(* IEC 61131-3 sources: F100R_S278_Temperville/MyController.device.xml.v3^/Plc Logic.plclogic.xml.v3^/Application.application.xml.v3^/00_FB, 42 files *)

(* ---- Valor_Float.fn.st ---- *)
FUNCTION Valor_Float : REAL
VAR_INPUT
	Input_01: WORD;
	Input_02: WORD;
END_VAR
VAR
	Convert_01: WORD_AS_DWORD;
	DW_AxOutpt: DWORD;
	Bit_DWord_Mantissa: BIT_AS_DWORD;
	Aux_Mantissa: DWORD;
	Mantissa1: REAL;
	Bit_DW_Expoente: BIT_AS_DWORD;
	Aux_Exp: DWORD;
	Aux_Exp2: REAL;
	Expoente: REAL;
	Sinal: REAL;
	Sinal2: REAL;
	base1: REAL;
END_VAR

Convert_01(i_wLow:= Input_01, i_wHigh:= Input_02, q_dwOput=>DW_AxOutpt );

(*=========== F=-1^s * 2^(e-127) * (1 + M/2^23)============= *)

//Composição da Mantissa
Bit_DWord_Mantissa(
	B00:= DW_AxOutpt.0,
	B01:= DW_AxOutpt.1,
	B02:= DW_AxOutpt.2,
	B03:= DW_AxOutpt.3,
	B04:= DW_AxOutpt.4,
	B05:= DW_AxOutpt.5,
	B06:= DW_AxOutpt.6,
	B07:= DW_AxOutpt.7,
	B08:= DW_AxOutpt.8,
	B09:= DW_AxOutpt.9,
	B10:= DW_AxOutpt.10,
	B11:= DW_AxOutpt.11,
	B12:= DW_AxOutpt.12,
	B13:= DW_AxOutpt.13,
	B14:= DW_AxOutpt.14,
	B15:= DW_AxOutpt.15,
	B16:= DW_AxOutpt.16,
	B17:= DW_AxOutpt.17,
	B18:= DW_AxOutpt.18,
	B19:= DW_AxOutpt.19,
	B20:= DW_AxOutpt.20,
	B21:= DW_AxOutpt.21,
	B22:= DW_AxOutpt.22,
	X=> Aux_Mantissa);

	Mantissa1:= DWORD_TO_REAL (Aux_Mantissa);

	//Composição Expoente

	Bit_DW_Expoente(
	B00:= DW_AxOutpt.23,
	B01:= DW_AxOutpt.24,
	B02:= DW_AxOutpt.25,
	B03:= DW_AxOutpt.26,
	B04:= DW_AxOutpt.27,
	B05:= DW_AxOutpt.28,
	B06:= DW_AxOutpt.29,
	B07:= DW_AxOutpt.30,
	X=> Aux_Exp);

	Aux_Exp2:= DWORD_TO_REAL (Aux_Exp - 127);

	Expoente:= EXPT (2,Aux_Exp2);

	//Sinal
	base1:=BOOL_TO_REAL (DW_AxOutpt.31);
	Sinal2:= EXPT (-1,base1);

	// Equação para o resultado em FLOAT

	Valor_Float:= Sinal2 * Expoente * (1 + Mantissa1/ 8388608);

(* ---- AlarmeEncoder.fb.st ---- *)
FUNCTION_BLOCK AlarmeEncoder
VAR_INPUT
	xHabilitaAlarme: BOOL;
	xResetAlarme: BOOL;
	ixCanalA: BOOL;
	ixCanalB: BOOL;
	tTempoPulso: TIME;
END_VAR
VAR_OUTPUT
	xAlarmeCanalA: BOOL;
	xAlarmeCanalB: BOOL;
	xAlarmeGeral: BOOL;
	xAlarmeSonoro: BOOL;
END_VAR
VAR
	TonAtrasoAlarme: TON;
	TonAtrasoAlarmeIn: BOOL;
	TonAtrasoAlarmePt: TIME;
	TonAtrasoAlarmeQ: BOOL;
	TonPulsoCanalAUp: TON;
	TonPulsoCanalAUpIn: BOOL;
	TonPulsoCanalAUpPt: TIME;
	TonPulsoCanalAUpQ: BOOL;
	TonPulsoCanalADown: TON;
	TonPulsoCanalADownIn: BOOL;
	TonPulsoCanalADownPt: TIME;
	TonPulsoCanalADownQ: BOOL;
	TonPulsoCanalBUp: TON;
	TonPulsoCanalBUpIn: BOOL;
	TonPulsoCanalBUpPt: TIME;
	TonPulsoCanalBUpQ: BOOL;
	TonPulsoCanalBDown: TON;
	TonPulsoCanalBDownIn: BOOL;
	TonPulsoCanalBDownPt: TIME;
	TonPulsoCanalBDownQ: BOOL;
	TonSinAlarme: TON;
	TonSinAlarmeIn: BOOL;
	TonSinAlarmePt: TIME;
	TonSinAlarmeQ: BOOL;
	TpSireneAlarme: TP;
	TpSireneAlarmeIn: BOOL;
	TpSireneAlarmePt: TIME;
	TpSireneAlarmeQ: BOOL;
	xHabilitadorMonitoraAlarme: BOOL;
END_VAR

(*Bloco de Monitoramento de Encoder pelas Entradas Digitais*)

(*---- Habilita Monitoramento de Alarme de Defeito ----*)
if xHabilitaAlarme then
	TonAtrasoAlarmeIn:=true;
else
	TonAtrasoAlarmeIn:=false;
end_if;

(*--- Tempo de Atraso para Inicio do Monitoramento ---*)
TonAtrasoAlarme (IN := TonAtrasoAlarmeIn,
		 PT := T#1500ms,
                 Q => TonAtrasoAlarmeQ);

xHabilitadorMonitoraAlarme:=TonAtrasoAlarmeQ;

(*--- Monitoramento do Canal A ---*)
(*--- Canal A Defeito Alto ---*)
TonPulsoCanalAUpIn:=xHabilitadorMonitoraAlarme and not ixCanalA;

TonPulsoCanalAUp (IN := TonPulsoCanalAUpIn,
                PT :=  tTempoPulso,
                Q => TonPulsoCanalAUpQ);

(*--- Canal A Defeito Baixo ---*)
TonPulsoCanalADownIn:=xHabilitadorMonitoraAlarme and ixCanalA;

TonPulsoCanalADown (IN := TonPulsoCanalADownIn,
                PT := tTempoPulso,
                Q => TonPulsoCanalADownQ);

(*--- Alarme Defeito Canal A ---*)

if TonPulsoCanalAUpQ or TonPulsoCanalADownQ then
	xAlarmeCanalA:=true;
end_if;

(*--------------------------------*)
(*--- Monitoramento do Canal B ---*)
(*--- Canal B Defeito Alto ---*)
TonPulsoCanalBUpIn:=xHabilitadorMonitoraAlarme and not ixCanalB;

TonPulsoCanalBUp (IN := TonPulsoCanalBUpIn,
                PT := tTempoPulso,
                Q => TonPulsoCanalBUpQ);

(*--- Canal A Defeito Baixo ---*)
TonPulsoCanalBDownIn:=xHabilitadorMonitoraAlarme and ixCanalB;

TonPulsoCanalBDown (IN := TonPulsoCanalBDownIn,
                PT := tTempoPulso,
                Q => TonPulsoCanalBDownQ);

(*--- Alarme Defeito Canal B ---*)

if TonPulsoCanalBUpQ or TonPulsoCanalBDownQ then
	xAlarmeCanalB:=true;
end_if;

(*--------------------------------*)
(*--- Indicação Alarme Geral ---*)
xAlarmeGeral:=xAlarmeCanalA or xAlarmeCanalB;

(*--- Alarme Sonoro ---*)
TpSireneAlarmeIn:=xAlarmeGeral;

TpSireneAlarme (IN := TpSireneAlarmeIn,
                PT := T#500ms,
                Q => TpSireneAlarmeQ);

if TpSireneAlarmeQ then
	xAlarmeSonoro:=true;
end_if;

(*--- Reseta Alarmes do Encoder ---*)
if xResetAlarme then
	xAlarmeCanalA:=false;
	xAlarmeCanalB:=false;
	xAlarmeSonoro:=false;
end_if;

(* ---- AlarmeMotor.fb.st ---- *)
FUNCTION_BLOCK AlarmeMotor
VAR_INPUT
	KaMotor: BOOL;
	KmMotor: BOOL;
	ResetAlarm: BOOL;
END_VAR
VAR_OUTPUT
	AlarmeMotor: BOOL;
	AlarmeSonoro: BOOL;
END_VAR
VAR
	TonAlarme: TON;
	TpSom: TP;
END_VAR

TonAlarme.IN:= KmMotor AND NOT KaMotor;

TonAlarme(PT:=T#100MS );

IF TonAlarme.Q THEN
	AlarmeMotor:= TRUE;
END_IF

TpSom(IN:= AlarmeMotor , PT:= T#500MS );

IF TpSom.Q THEN
	AlarmeSonoro:=TRUE;
END_IF

IF	ResetAlarm THEN
	AlarmeMotor:=FALSE;
	AlarmeSonoro:=FALSE;
END_IF

(* ---- AlarmeMotorParado.fb.st ---- *)
FUNCTION_BLOCK AlarmeMotorParado
VAR_INPUT
	KaMotor: BOOL;
	ResetAlarm: BOOL;
END_VAR
VAR_OUTPUT
	AlarmeMotor: BOOL;
	AlarmeSonoro: BOOL;
END_VAR
VAR
	TonAlarme: TON;
	TpSom: TP;
	TpReset: TP;
END_VAR

TonAlarme.IN:= KaMotor;

TonAlarme(PT:=T#3000MS );

IF TonAlarme.Q THEN
	AlarmeMotor:= TRUE;
END_IF

TpSom(IN:= AlarmeMotor , PT:= T#500MS );

IF TpSom.Q THEN
	AlarmeSonoro:=TRUE;
END_IF

TpReset(IN:= ResetAlarm , PT:= T#1000MS );

IF	TpReset.Q THEN
	AlarmeMotor:=FALSE;
	AlarmeSonoro:=FALSE;
END_IF

(* ---- AlarmeRelesSsr.fb.st ---- *)
FUNCTION_BLOCK AlarmeRelesSsr
VAR_INPUT
	RetornoReleSsr: BOOL;
	ResistRompida: BOOL;
	ReleSsr: BOOL;
	ResetAlarm: BOOL;
END_VAR
VAR_OUTPUT
	AlarmeSsrAberto: BOOL;
	AlarmeSsrFechado: BOOL;
	AlarmeSonoro: BOOL;
END_VAR
VAR
	TonAberto: TON;
	TonFechado: TON;
	TpSom: TP;
END_VAR

TonAberto.IN:= ReleSsr AND NOT RetornoReleSsr;
TonFechado.IN:= RetornoReleSsr AND NOT ResistRompida AND NOT ReleSsr;

TonAberto(PT:=T#400MS );
TonFechado(PT:=T#400MS );

IF TonAberto.Q THEN
	AlarmeSsrAberto:= TRUE;
END_IF

IF TonFechado.Q THEN
	AlarmeSsrFechado:=TRUE;
END_IF

TpSom(IN:= AlarmeSsrAberto OR AlarmeSsrFechado, PT:= T#200MS );

IF TpSom.Q THEN
	AlarmeSonoro:=TRUE;
END_IF

IF	ResetAlarm THEN
	AlarmeSsrAberto:=FALSE;
	AlarmeSsrFechado:=FALSE;
	AlarmeSonoro:=FALSE;
END_IF

(* ---- AlarmeResistencia.fb.st ---- *)
FUNCTION_BLOCK AlarmeResistencia
VAR_INPUT
	ResistRompida: BOOL;
	ResetAlarm: BOOL;
END_VAR
VAR_OUTPUT
	AlarmeResistRompida: BOOL;
	AlarmeSonoro: BOOL;
END_VAR
VAR
	TonRompida: TON;
	TpSom: TP;
END_VAR

TonRompida.IN:=ResistRompida;

TonRompida(PT:=T#250ms);

IF TonRompida.Q THEN
	AlarmeResistRompida:=TRUE;
END_IF

TpSom(IN:= AlarmeResistRompida, PT:= T#500MS);

IF TpSom.Q THEN
	AlarmeSonoro:=TRUE;
END_IF

IF	ResetAlarm THEN
	AlarmeResistRompida:=FALSE;
	AlarmeSonoro:=FALSE;
END_IF

(* ---- AlarmeTemperatura.fb.st ---- *)
FUNCTION_BLOCK AlarmeTemperatura
VAR_INPUT
	TermoparAtual: REAL;
	TemperaturaMax: REAL;
	ResetAlarm: BOOL;
END_VAR
VAR_OUTPUT
	TermoparAlmTemperatura: BOOL;
	AlarmeSonAlmTemperatura: BOOL;
END_VAR
VAR
	TonTh: TON;
	TpSom: TP;
	TemperaturaExcedeu: BOOL;
END_VAR

TemperaturaExcedeu:=(TermoparAtual >= TemperaturaMax);

TonTh.IN:=TemperaturaExcedeu;

TonTh(PT:=T#1S);

IF TonTh.Q THEN
	TermoparAlmTemperatura:=TRUE;
END_IF

TpSom(IN:=TermoparAlmTemperatura,PT:=T#1S);

IF TpSom.Q THEN
	AlarmeSonAlmTemperatura:=TRUE;
END_IF

IF	ResetAlarm THEN
	TermoparAlmTemperatura:=FALSE;
	AlarmeSonAlmTemperatura:=FALSE;
END_IF

(* ---- AlarmeTermopar.fb.st ---- *)
FUNCTION_BLOCK AlarmeTermopar
VAR_INPUT
	Termopar: BOOL;
	ResetAlarm: BOOL;
END_VAR
VAR_OUTPUT
	TermoparAberto: BOOL;
	AlarmeSonTermopar: BOOL;
END_VAR
VAR
	TonTh: TON;
	TpSom: TP;
END_VAR

TonTh.IN:=Termopar;

TonTh(PT:=T#1S);

IF TonTh.Q THEN
	TermoparAberto:=TRUE;
END_IF

TpSom(IN:=TermoparAberto,PT:=T#1S);

IF TpSom.Q THEN
	AlarmeSonTermopar:=TRUE;
END_IF

IF	ResetAlarm THEN
	TermoparAberto:=FALSE;
	AlarmeSonTermopar:=FALSE;
END_IF

(* ---- AlarmeTM3TI8T.fb.st ---- *)
FUNCTION_BLOCK AlarmeTM3TI8T
VAR_INPUT
	inAlarmeInput01: BYTE;
	inAlarmeInput02: BYTE;
	inAlarmeInput03: BYTE;
	inAlarmeInput04: BYTE;
	inAlarmeInput05: BYTE;
	inAlarmeInput06: BYTE;
	inAlarmeInput07: BYTE;
	inAlarmeInput08: BYTE;
END_VAR
VAR_OUTPUT
	OutAlarmeInput01: BOOL;
	OutAlarmeInput02: BOOL;
	OutAlarmeInput03: BOOL;
	OutAlarmeInput04: BOOL;
	OutAlarmeInput05: BOOL;
	OutAlarmeInput06: BOOL;
	OutAlarmeInput07: BOOL;
	OutAlarmeInput08: BOOL;
END_VAR
VAR
	TonTh01: TON;
	TonTh02: TON;
	TonTh03: TON;
	TonTh04: TON;
	TonTh05: TON;
	TonTh06: TON;
	TonTh07: TON;
	TonTh08: TON;
	xTermopar01Aberto: BOOL;
	xTermopar02Aberto: BOOL;
	xTermopar03Aberto: BOOL;
	xTermopar04Aberto: BOOL;
	xTermopar05Aberto: BOOL;
	xTermopar06Aberto: BOOL;
	xTermopar07Aberto: BOOL;
	xTermopar08Aberto: BOOL;
END_VAR

//TERMOPAR 01
IF inAlarmeInput01=5 OR inAlarmeInput01=6 OR inAlarmeInput01=4 THEN
	xTermopar01Aberto:=TRUE;
ELSE
	xTermopar01Aberto:=FALSE;
END_IF

//TERMOPAR 02
IF inAlarmeInput02=5 OR inAlarmeInput02=6 OR inAlarmeInput02=4 THEN
	xTermopar02Aberto:=TRUE;
ELSE
	xTermopar02Aberto:=FALSE;
END_IF

//TERMOPAR 03
IF inAlarmeInput03=5 OR inAlarmeInput03=6 OR inAlarmeInput03=4 THEN
	xTermopar03Aberto:=TRUE;
ELSE
	xTermopar03Aberto:=FALSE;
END_IF

//TERMOPAR 04
IF inAlarmeInput04=5 OR inAlarmeInput04=6 OR inAlarmeInput04=4 THEN
	xTermopar04Aberto:=TRUE;
ELSE
	xTermopar04Aberto:=FALSE;
END_IF

//TERMOPAR 05
IF inAlarmeInput05=5 OR inAlarmeInput05=6 OR inAlarmeInput05=4 THEN
	xTermopar05Aberto:=TRUE;
ELSE
	xTermopar05Aberto:=FALSE;
END_IF

//TERMOPAR 06
IF inAlarmeInput06=5 OR inAlarmeInput06=6 OR inAlarmeInput06=4 THEN
	xTermopar06Aberto:=TRUE;
ELSE
	xTermopar06Aberto:=FALSE;
END_IF

//TERMOPAR 07
IF inAlarmeInput07=5 OR inAlarmeInput07=6 OR inAlarmeInput07=4 THEN
	xTermopar07Aberto:=TRUE;
ELSE
	xTermopar07Aberto:=FALSE;
END_IF

//TERMOPAR 08
IF inAlarmeInput08=5 OR inAlarmeInput08=6 OR inAlarmeInput08=4 THEN
	xTermopar08Aberto:=TRUE;
ELSE
	xTermopar08Aberto:=FALSE;
END_IF

TonTh01(IN:=xTermopar01Aberto, PT:=T#0S , Q=>OutAlarmeInput01);
TonTh02(IN:=xTermopar02Aberto, PT:=T#0S , Q=>OutAlarmeInput02);
TonTh03(IN:=xTermopar03Aberto, PT:=T#0S , Q=>OutAlarmeInput03);
TonTh04(IN:=xTermopar04Aberto, PT:=T#0S , Q=>OutAlarmeInput04);
TonTh05(IN:=xTermopar05Aberto, PT:=T#0S , Q=>OutAlarmeInput05);
TonTh06(IN:=xTermopar06Aberto, PT:=T#0S , Q=>OutAlarmeInput06);
TonTh07(IN:=xTermopar07Aberto, PT:=T#0S , Q=>OutAlarmeInput07);
TonTh08(IN:=xTermopar08Aberto, PT:=T#0S , Q=>OutAlarmeInput08);

(* ---- AlarmeTM5SAI6TH.fb.st ---- *)
FUNCTION_BLOCK AlarmeTM5SAI6TH
VAR_INPUT
	bEntradaByte00: BYTE;
	bEntradaByte01: BYTE;
	ResetAlarm: BOOL;
END_VAR
VAR_OUTPUT
	Termopar01AbaixoMinimo: BOOL;
	Termopar01AcimaMaximo: BOOL;
	Termopar01Ok: BOOL;
	Termopar01Aberto: BOOL;
	Termopar02AbaixoMinimo: BOOL;
	Termopar02AcimaMaximo: BOOL;
	Termopar02Ok: BOOL;
	Termopar02Aberto: BOOL;
	Termopar03AbaixoMinimo: BOOL;
	Termopar03AcimaMaximo: BOOL;
	Termopar03Ok: BOOL;
	Termopar03Aberto: BOOL;
	Termopar04AbaixoMinimo: BOOL;
	Termopar04AcimaMaximo: BOOL;
	Termopar04Ok: BOOL;
	Termopar04Aberto: BOOL;
	Termopar05AbaixoMinimo: BOOL;
	Termopar05AcimaMaximo: BOOL;
	Termopar05Ok: BOOL;
	Termopar05Aberto: BOOL;
	Termopar06AbaixoMinimo: BOOL;
	Termopar06AcimaMaximo: BOOL;
	Termopar06Ok: BOOL;
	Termopar06Aberto: BOOL;
END_VAR
VAR
	StatusByte00: BYTE_AS_BIT;
	StatusByte01: BYTE_AS_BIT;
	xEntradaTermopar0101: BOOL;
	xEntradaTermopar0201: BOOL;
	xEntradaTermopar0102: BOOL;
	xEntradaTermopar0202: BOOL;
	xEntradaTermopar0103: BOOL;
	xEntradaTermopar0203: BOOL;
	xEntradaTermopar0104: BOOL;
	xEntradaTermopar0204: BOOL;
	xEntradaTermopar0105: BOOL;
	xEntradaTermopar0205: BOOL;
	xEntradaTermopar0106: BOOL;
	xEntradaTermopar0206: BOOL;
	TonTh01: TON;
	TonTh02: TON;
	TonTh03: TON;
	TonTh04: TON;
	TonTh05: TON;
	TonTh06: TON;
END_VAR

StatusByte00(
		B:= bEntradaByte00,
		B0=> xEntradaTermopar0101,
		B1=> xEntradaTermopar0201,
		B2=> xEntradaTermopar0102,
		B3=> xEntradaTermopar0202,
		B4=> xEntradaTermopar0103,
		B5=> xEntradaTermopar0203,
		B6=> xEntradaTermopar0104,
		B7=> xEntradaTermopar0204);

StatusByte01(
		B:= bEntradaByte01,
		B0=> xEntradaTermopar0105,
		B1=> xEntradaTermopar0205,
		B2=> xEntradaTermopar0106,
		B3=> xEntradaTermopar0206);

Termopar01Ok:= NOT xEntradaTermopar0101 AND NOT xEntradaTermopar0201;
Termopar01AbaixoMinimo:= NOT xEntradaTermopar0101 AND xEntradaTermopar0201;
Termopar01AcimaMaximo:= xEntradaTermopar0101 AND NOT xEntradaTermopar0201;
TonTh01.IN:= xEntradaTermopar0101 AND xEntradaTermopar0201;

Termopar02Ok:= NOT xEntradaTermopar0102 AND NOT xEntradaTermopar0202;
Termopar02AbaixoMinimo:= NOT xEntradaTermopar0102 AND xEntradaTermopar0202;
Termopar02AcimaMaximo:= xEntradaTermopar0102 AND NOT xEntradaTermopar0202;
TonTh02.IN:= xEntradaTermopar0102 AND xEntradaTermopar0202;

Termopar03Ok:= NOT xEntradaTermopar0103 AND NOT xEntradaTermopar0203;
Termopar03AbaixoMinimo:= NOT xEntradaTermopar0103 AND xEntradaTermopar0203;
Termopar03AcimaMaximo:= xEntradaTermopar0103 AND NOT xEntradaTermopar0203;
TonTh03.IN:= xEntradaTermopar0103 AND xEntradaTermopar0203;

Termopar04Ok:= NOT xEntradaTermopar0104 AND NOT xEntradaTermopar0204;
Termopar04AbaixoMinimo:= NOT xEntradaTermopar0104 AND xEntradaTermopar0204;
Termopar04AcimaMaximo:= xEntradaTermopar0104 AND NOT xEntradaTermopar0204;
TonTh04.IN:= xEntradaTermopar0104 AND xEntradaTermopar0204;

Termopar05Ok:= NOT xEntradaTermopar0105 AND NOT xEntradaTermopar0205;
Termopar05AbaixoMinimo:= NOT xEntradaTermopar0105 AND xEntradaTermopar0205;
Termopar05AcimaMaximo:= xEntradaTermopar0105 AND NOT xEntradaTermopar0205;
TonTh05.IN:= xEntradaTermopar0105 AND xEntradaTermopar0205;

Termopar06Ok:= NOT xEntradaTermopar0106 AND NOT xEntradaTermopar0206;
Termopar06AbaixoMinimo:= NOT xEntradaTermopar0106 AND xEntradaTermopar0206;
Termopar06AcimaMaximo:= xEntradaTermopar0106 AND NOT xEntradaTermopar0206;
TonTh06.IN:= xEntradaTermopar0106 AND xEntradaTermopar0206;

TonTh01(PT:=T#0S , Q=>Termopar01Aberto);
TonTh02(PT:=T#0S , Q=>Termopar02Aberto);
TonTh03(PT:=T#0S , Q=>Termopar03Aberto);
TonTh04(PT:=T#0S , Q=>Termopar04Aberto);
TonTh05(PT:=T#0S , Q=>Termopar05Aberto);
TonTh06(PT:=T#0S , Q=>Termopar06Aberto);

(* ---- AlarmeValvula1v.fb.st ---- *)
FUNCTION_BLOCK AlarmeValvula1v
VAR_INPUT
	SensorValvAberta: BOOL;
	SensorValvFechad: BOOL;
	AcionamentoValvula: BOOL;
	ResetAlarm: BOOL;
	TempoAberto: TIME;
	TempoFechad: TIME;
END_VAR
VAR_OUTPUT
	AlarmeValvAberta: BOOL;
	AlarmeValvFechada: BOOL;
	AlarmeSonoro: BOOL;
END_VAR
VAR
	TonAberto: TON;
	TonFechado: TON;
	TpSom: TP;
END_VAR

TonAberto.IN:= AcionamentoValvula AND NOT SensorValvAberta;
TonFechado.IN:= NOT AcionamentoValvula AND NOT SensorValvFechad;

TonAberto(PT:= TempoAberto);
TonFechado(PT:=TempoFechad );

IF TonAberto.Q THEN
	AlarmeValvAberta:= TRUE;
END_IF

IF TonFechado.Q THEN
	AlarmeValvFechada:=TRUE;
END_IF

TpSom(IN:= AlarmeValvAberta OR AlarmeValvFechada, PT:= T#500MS );

IF TpSom.Q THEN
	AlarmeSonoro:=TRUE;
END_IF

IF	ResetAlarm THEN
	AlarmeValvAberta:=FALSE;
	AlarmeValvFechada:=FALSE;
	AlarmeSonoro:=FALSE;
END_IF

(* ---- AlarmeValvula1vNeg.fb.st ---- *)
FUNCTION_BLOCK AlarmeValvula1vNeg
VAR_INPUT
	SensorValvAberta: BOOL;
	SensorValvFechad: BOOL;
	AcionamentoValvula: BOOL;
	ResetAlarm: BOOL;
	TempoAberto: TIME;
	TempoFechad: TIME;
END_VAR
VAR_OUTPUT
	AlarmeValvAberta: BOOL;
	AlarmeValvFechada: BOOL;
	AlarmeSonoro: BOOL;
END_VAR
VAR
	TonAberto: TON;
	TonFechado: TON;
	TpSom: TP;
END_VAR

TonAberto.IN:= NOT AcionamentoValvula AND NOT SensorValvAberta;
TonFechado.IN:= AcionamentoValvula AND NOT SensorValvFechad;

TonAberto(PT:= TempoAberto);
TonFechado(PT:=TempoFechad );

IF TonAberto.Q THEN
	AlarmeValvAberta:= TRUE;
END_IF

IF TonFechado.Q THEN
	AlarmeValvFechada:=TRUE;
END_IF

TpSom(IN:= AlarmeValvAberta OR AlarmeValvFechada, PT:= T#500MS );

IF TpSom.Q THEN
	AlarmeSonoro:=TRUE;
END_IF

IF	ResetAlarm THEN
	AlarmeValvAberta:=FALSE;
	AlarmeValvFechada:=FALSE;
	AlarmeSonoro:=FALSE;
END_IF

(* ---- BlocoSelecaoEspessura.fb.st ---- *)
FUNCTION_BLOCK BlocoSelecaoEspessura
VAR_INPUT
	xSelecao: BOOL;
	iEntrada0101: INT;
	iEntrada0102: INT;
	iEntrada0201: INT;
	iEntrada0202: INT;
	iEntrada0301: INT;
	iEntrada0302: INT;
	iEntrada0401: INT;
	iEntrada0402: INT;
	iEntrada0501: INT;
	iEntrada0502: INT;
	iEntrada0601: INT;
	iEntrada0602: INT;
	iEntrada0701: INT;
	iEntrada0702: INT;
	iEntrada0801: INT;
	iEntrada0802: INT;
	iEntrada0901: INT;
	iEntrada0902: INT;
	iEntrada1001: INT;
	iEntrada1002: INT;
END_VAR
VAR_OUTPUT
	iSaida01: INT;
	iSaida02: INT;
	iSaida03: INT;
	iSaida04: INT;
	iSaida05: INT;
	iSaida06: INT;
	iSaida07: INT;
	iSaida08: INT;
	iSaida09: INT;
	iSaida10: INT;
END_VAR
VAR
	SelecaoEspessuraParam01: SelecaoEspessura;
	SelecaoEspessuraParam02: SelecaoEspessura;
	SelecaoEspessuraParam03: SelecaoEspessura;
	SelecaoEspessuraParam04: SelecaoEspessura;
	SelecaoEspessuraParam05: SelecaoEspessura;
	SelecaoEspessuraParam06: SelecaoEspessura;
	SelecaoEspessuraParam07: SelecaoEspessura;
	SelecaoEspessuraParam08: SelecaoEspessura;
	SelecaoEspessuraParam09: SelecaoEspessura;
	SelecaoEspessuraParam10: SelecaoEspessura;
END_VAR

SelecaoEspessuraParam01(Selecao:=xSelecao , Entrada01:=iEntrada0101 , Entrada02:=iEntrada0102 , Saida=>iSaida01 );
SelecaoEspessuraParam02(Selecao:=xSelecao , Entrada01:=iEntrada0201 , Entrada02:=iEntrada0202 , Saida=>iSaida02 );
SelecaoEspessuraParam03(Selecao:=xSelecao , Entrada01:=iEntrada0301 , Entrada02:=iEntrada0302 , Saida=>iSaida03 );
SelecaoEspessuraParam04(Selecao:=xSelecao , Entrada01:=iEntrada0401 , Entrada02:=iEntrada0402 , Saida=>iSaida04 );
SelecaoEspessuraParam05(Selecao:=xSelecao , Entrada01:=iEntrada0501 , Entrada02:=iEntrada0502 , Saida=>iSaida05 );
SelecaoEspessuraParam06(Selecao:=xSelecao , Entrada01:=iEntrada0601 , Entrada02:=iEntrada0602 , Saida=>iSaida06 );
SelecaoEspessuraParam07(Selecao:=xSelecao , Entrada01:=iEntrada0701 , Entrada02:=iEntrada0702 , Saida=>iSaida07 );
SelecaoEspessuraParam08(Selecao:=xSelecao , Entrada01:=iEntrada0801 , Entrada02:=iEntrada0802 , Saida=>iSaida08 );
SelecaoEspessuraParam09(Selecao:=xSelecao , Entrada01:=iEntrada0901 , Entrada02:=iEntrada0902 , Saida=>iSaida09 );
SelecaoEspessuraParam10(Selecao:=xSelecao , Entrada01:=iEntrada1001 , Entrada02:=iEntrada1002 , Saida=>iSaida10 );

(* ---- CalculosForno.fb.st ---- *)
FUNCTION_BLOCK CalculosForno
VAR_INPUT
	DistanciaVelMinForno: INT;
	DistanciaCargaForno: INT;
	TamanhoAreaUtil: INT;
	TamanhoCargaMaxima: INT;
	TamanhoCarga: INT;
END_VAR
VAR_OUTPUT
	SetPointVelMinCarga: INT;
	SetPointCargaForno: INT;
	SetPointDescargaForno: INT;
	SetPointAvancaVaiVemForno: INT;
	SetPointRecuaVaiVemForno: INT;
	TamanhoAreaUtilForno: INT;
	TamanhoCargaMaxForno: INT;
END_VAR

SetPointVelMinCarga:= DistanciaCargaForno-DistanciaVelMinForno;
SetPointCargaForno:= DistanciaCargaForno;
SetPointDescargaForno:= DistanciaCargaForno+TamanhoAreaUtil;
SetPointAvancaVaiVemForno:= DistanciaCargaForno;
SetPointRecuaVaiVemForno:= DistanciaCargaForno-(TamanhoAreaUtilForno-TamanhoCarga);
TamanhoAreaUtilForno:= TamanhoAreaUtil;
TamanhoCargaMaxForno := TamanhoCargaMaxima;

(* ---- CalculosResfriador.fb.st ---- *)
FUNCTION_BLOCK CalculosResfriador
VAR_INPUT
	DistanciaVelMinResfriador: INT;
	DistanciaCargaResfriador: INT;
	DistanciaOscilacaoResfriador: INT;
	DistanciaDescargaResfriador: INT;
	TamanhoAreaUtil: INT;
	///////
	TamanhoCarga: INT;
END_VAR
VAR_OUTPUT
	SetPointVelMinCarga: INT;
	SetPointCargaResfriador: INT;
	SetPointDescargaResfriador: INT;
	SetPointAvancaVaiVemResfriador: INT;
	SetPointRecuaVaiVemResfriador: INT;
END_VAR

(*SetPointVelMinCarga:= DistanciaCargaResfriador-DistanciaVelMinResfriador;
SetPointCargaResfriador:= DistanciaCargaResfriador;
SetPointDescargaResfriador:= DistanciaDescargaResfriador;
SetPointAvancaVaiVemResfriador:= DistanciaCargaResfriador;
SetPointRecuaVaiVemResfriador:= DistanciaCargaResfriador-DistanciaOscilacaoResfriador;*)

SetPointVelMinCarga:= DistanciaCargaResfriador-DistanciaVelMinResfriador;
SetPointCargaResfriador:= DistanciaCargaResfriador;
SetPointDescargaResfriador:= DistanciaDescargaResfriador;
SetPointAvancaVaiVemResfriador:= DistanciaCargaResfriador;
SetPointRecuaVaiVemResfriador:= DistanciaCargaResfriador-(TamanhoAreaUtil-TamanhoCarga);

(* ---- ComprimentoCarga.fb.st ---- *)
FUNCTION_BLOCK ComprimentoCarga
VAR_INPUT
	Sensor: BOOL;
	Habilita: BOOL;
	ValEncoder: DINT;
END_VAR
VAR_OUTPUT
	TamanhoCarga: DINT;
END_VAR
VAR_IN_OUT
	FimMedicao: BOOL;
END_VAR
VAR
	PulsoSensorNe: PulsoNegativo;
	PulsoSensorPo: PulsoPositivo;
	PulsoHabilitaNe: PulsoNegativo;
	PulsoHabilitaPo: PulsoPositivo;
	TamanhoCargaAux: DINT;
END_VAR

PulsoSensorNe(Entrada:= Sensor, SaidaPulsoNe=> );
PulsoSensorPo(Entrada:= Sensor, SaidaPulsoPo=> );

IF PulsoSensorNe.SaidaPulsoNe OR PulsoSensorPo.SaidaPulsoPo THEN
	TamanhoCargaAux:= ValEncoder;
END_IF

PulsoHabilitaPo(Entrada:= Habilita, SaidaPulsoPo=>);

IF PulsoHabilitaPo.SaidaPulsoPo THEN
	TamanhoCargaAux:=0;
END_IF

PulsoHabilitaNe(Entrada:= Habilita, SaidaPulsoNe=> );

IF PulsoHabilitaNe.SaidaPulsoNe THEN
	TamanhoCarga:=TamanhoCargaAux;
	FimMedicao:=TRUE;
END_IF

(* ---- ContadorUpDown.fb.st ---- *)
FUNCTION_BLOCK ContadorUpDown
VAR_INPUT
	CU: BOOL;
	CD: BOOL;
	RESET: BOOL;
END_VAR
VAR_OUTPUT
	CV: INT;
END_VAR
VAR
	PulsoSobe: PulsoPositivo;
	PulsoDesc: PulsoPositivo;
	PulsoSobeSaida: BOOL;
	PulsoDescSaida: BOOL;
END_VAR

PulsoSobe(Entrada:=CU , SaidaPulsoPo=>PulsoSobeSaida );
PulsoDesc(Entrada:=CD , SaidaPulsoPo=>PulsoDescSaida );

IF PulsoSobeSaida THEN
	CV:=CV+1;
END_IF
IF PulsoDescSaida THEN
	CV:=CV-1;
END_IF
IF RESET THEN
	CV:=0;
END_IF

(* ---- EncoderBlocoExpert.fb.st ---- *)
FUNCTION_BLOCK EncoderBlocoExpert
VAR_INPUT
	Entrada: DINT;
	Zera: BOOL;
	InversaoSinal: BOOL;
END_VAR
VAR_OUTPUT
	Contagem: DINT;
END_VAR
VAR
	ValorZera: DINT := 0;
	Valor: DINT;
END_VAR

IF Zera THEN
	ValorZera:=Entrada;
END_IF

Valor:=Entrada-ValorZera;

IF InversaoSinal THEN
	Contagem:=-1*Valor;
ELSE
	Contagem:=Valor;
END_IF

(* ---- EquacaoDaReta.fb.st ---- *)
FUNCTION_BLOCK EquacaoDaReta
VAR_INPUT
	rValorY: REAL;
	rPy1: REAL;
	rPy2: REAL;
	rPx1: REAL;
	rPx2: REAL;
END_VAR
VAR_OUTPUT
	rValorX: REAL;
END_VAR
VAR
	Aux01: REAL;
	Aux02: REAL;
	Aux03: REAL;
	Aux04: REAL;
	Aux05: REAL;
END_VAR

// EQUAÇÃO FUNDAMENTAL DA RETA

//X= (-Y*x2+Y*x1)-(x1*y2)+(y1*x2)/(y1-y2);

rValorX:= (-(rValorY*rPx2)+(rValorY*rPx1)-(rPx1*rPy2)+(rPy1*rPx2))/(rPy1-rPy2);

Aux01:=(rValorY*rPx2);
Aux02:=(rValorY*rPx1);
Aux03:=(rPx1*rPy2);
Aux04:=(rPy1*rPx2);
Aux05:=(rPy1-rPy2);

(* ---- Grade.fb.st ---- *)
FUNCTION_BLOCK Grade
VAR_IN_OUT
	LigaDesl: BOOL;
END_VAR
VAR_INPUT
	Libera: BOOL;
	Liga: BOOL;
	Desl: BOOL;
	Alarme01: BOOL;
END_VAR
VAR_OUTPUT
	StatusSaida: BOOL;
END_VAR
VAR
	PulsoHabilita: PulsoPositivo;
	PulsoHabilitaSaida: BOOL;
	Auxiliar01Habilita: BOOL;
	Auxiliar02Habilita: BOOL;
END_VAR

PulsoHabilita(Entrada:=LigaDesl , SaidaPulsoPo=> PulsoHabilitaSaida);
Auxiliar02Habilita:=PulsoHabilitaSaida AND Auxiliar01Habilita AND Libera;
Auxiliar01Habilita:=(((PulsoHabilitaSaida OR (Liga AND Libera)) AND NOT  Auxiliar01Habilita) OR Auxiliar01Habilita) AND NOT Auxiliar02Habilita AND NOT (Desl AND Libera) AND NOT Alarme01;
StatusSaida:=Auxiliar01Habilita;

(* ---- HabilitaDesabilita.fb.st ---- *)
FUNCTION_BLOCK HabilitaDesabilita
VAR_IN_OUT
	Entrada: BOOL;
END_VAR
VAR_INPUT
	Entrada02: BOOL;
	Entrada03: BOOL;
	Alarme01: BOOL;
	Alarme02: BOOL;
	Alarme03: BOOL;
END_VAR
VAR_OUTPUT
	StatusSaida: BOOL;
END_VAR
VAR
	PulsoHabilita: PulsoPositivo;
	PulsoHabilitaSaida: BOOL;
	Auxiliar01Habilita: BOOL;
	Auxiliar02Habilita: BOOL;
END_VAR

PulsoHabilita(Entrada:=Entrada , SaidaPulsoPo=> PulsoHabilitaSaida);
Auxiliar02Habilita:=PulsoHabilitaSaida AND Auxiliar01Habilita;
Auxiliar01Habilita:=(((PulsoHabilitaSaida OR Entrada02) AND NOT  Auxiliar01Habilita) OR Auxiliar01Habilita) AND NOT Auxiliar02Habilita AND NOT Entrada03 AND NOT Alarme01 AND NOT Alarme02 AND NOT Alarme03;
StatusSaida:=Auxiliar01Habilita;
//Entrada := FALSE;

(* ---- HabilitaDesabilitaSB.fb.st ---- *)
FUNCTION_BLOCK HabilitaDesabilitaSB
VAR_IN_OUT
	Entrada: BOOL;
END_VAR
VAR_INPUT
	Entrada02: BOOL;
	Entrada03: BOOL;
	Alarme01: BOOL;
	Alarme02: BOOL;
	Alarme03: BOOL;
END_VAR
VAR_OUTPUT
	StatusSaida: BOOL;
END_VAR
VAR
	PulsoHabilita: PulsoPositivo;
	PulsoHabilitaSaida: BOOL;
	Auxiliar01Habilita: BOOL;
	Auxiliar02Habilita: BOOL;
END_VAR

PulsoHabilita(Entrada:=Entrada , SaidaPulsoPo=> PulsoHabilitaSaida);
Auxiliar02Habilita:=PulsoHabilitaSaida AND Auxiliar01Habilita;
Auxiliar01Habilita:=(((PulsoHabilitaSaida OR Entrada02) AND NOT  Auxiliar01Habilita) OR Auxiliar01Habilita) AND NOT Auxiliar02Habilita AND NOT Entrada03 AND NOT Alarme01 AND NOT Alarme02 AND NOT Alarme03;
StatusSaida:=Auxiliar01Habilita;
Entrada := FALSE;

(* ---- MmConversorPulso.fb.st ---- *)
FUNCTION_BLOCK MmConversorPulso
VAR_INPUT
	dPulso	: DINT;
	dMilimetro : DINT;
	iEntrMilimetro01: INT;
	iEntrMilimetro02: INT;
	iEntrMilimetro03: INT;
	iEntrMilimetro04: INT;
	iEntrMilimetro05: INT;
	iEntrMilimetro06: INT;
	iEntrMilimetro07: INT;
	iEntrMilimetro08: INT;
	iEntrMilimetro09: INT;
	iEntrMilimetro10: INT;
	iEntrMilimetro11: INT;
	iEntrMilimetro12: INT;
	iEntrMilimetro13: INT;
	iEntrMilimetro14: INT;
	iEntrMilimetro15: INT;
	iEntrMilimetro16: INT;
	iEntrMilimetro17: INT;
	iEntrMilimetro18: INT;
	iEntrMilimetro19: INT;
	iEntrMilimetro20: INT;
END_VAR
VAR_OUTPUT
	dSaidaPulso01:	DINT;
	dSaidaPulso02:	DINT;
	dSaidaPulso03:	DINT;
	dSaidaPulso04:	DINT;
	dSaidaPulso05:	DINT;
	dSaidaPulso06:	DINT;
	dSaidaPulso07:	DINT;
	dSaidaPulso08:	DINT;
	dSaidaPulso09:	DINT;
	dSaidaPulso10:	DINT;
	dSaidaPulso11:	DINT;
	dSaidaPulso12:	DINT;
	dSaidaPulso13:	DINT;
	dSaidaPulso14:	DINT;
	dSaidaPulso15:	DINT;
	dSaidaPulso16:	DINT;
	dSaidaPulso17:	DINT;
	dSaidaPulso18:	DINT;
	dSaidaPulso19:	DINT;
	dSaidaPulso20:	DINT;
END_VAR
VAR
	dEntrMilimetro03	: DINT ;
	dPulsodEntrMilimetro03	: DINT ;

	rEntrMilimetro03	: REAL ;
	rPulso				: REAL ;
	rMilimetro			: REAL ;
	rSaidaPulso03		: REAL ;
	rPulsodEntrMilimetro03	: real ;
END_VAR

rPulso:=DINT_TO_REAL(dPulso);
rMilimetro:=DINT_TO_REAL(dMilimetro);

dSaidaPulso01:=(dPulso*INT_TO_DINT(iEntrMilimetro01))/dMilimetro;
dSaidaPulso02:=(dPulso*INT_TO_DINT(iEntrMilimetro02))/dMilimetro;

dEntrMilimetro03:= INT_TO_DINT (iEntrMilimetro03);
rEntrMilimetro03:=DINT_TO_REAL(dEntrMilimetro03);

dPulsodEntrMilimetro03:=(dPulso*dEntrMilimetro03);
rPulsodEntrMilimetro03:=(rPulso*rEntrMilimetro03);

//dSaidaPulso03:=dPulsodEntrMilimetro03/dMilimetro;
rSaidaPulso03:=rPulsodEntrMilimetro03/rMilimetro;
dSaidaPulso03:=REAL_TO_DINT(rSaidaPulso03);

dSaidaPulso04:=(dPulso*INT_TO_DINT(iEntrMilimetro04))/dMilimetro;
dSaidaPulso05:=(dPulso*INT_TO_DINT(iEntrMilimetro05))/dMilimetro;
dSaidaPulso06:=(dPulso*INT_TO_DINT(iEntrMilimetro06))/dMilimetro;
dSaidaPulso07:=(dPulso*INT_TO_DINT(iEntrMilimetro07))/dMilimetro;
dSaidaPulso08:=(dPulso*INT_TO_DINT(iEntrMilimetro08))/dMilimetro;
dSaidaPulso09:=(dPulso*INT_TO_DINT(iEntrMilimetro09))/dMilimetro;
dSaidaPulso10:=(dPulso*INT_TO_DINT(iEntrMilimetro10))/dMilimetro;
dSaidaPulso11:=(dPulso*INT_TO_DINT(iEntrMilimetro11))/dMilimetro;
dSaidaPulso12:=(dPulso*INT_TO_DINT(iEntrMilimetro12))/dMilimetro;
dSaidaPulso13:=(dPulso*INT_TO_DINT(iEntrMilimetro13))/dMilimetro;
dSaidaPulso14:=(dPulso*INT_TO_DINT(iEntrMilimetro14))/dMilimetro;
dSaidaPulso15:=(dPulso*INT_TO_DINT(iEntrMilimetro15))/dMilimetro;
dSaidaPulso16:=(dPulso*INT_TO_DINT(iEntrMilimetro16))/dMilimetro;
dSaidaPulso17:=(dPulso*INT_TO_DINT(iEntrMilimetro17))/dMilimetro;
dSaidaPulso18:=(dPulso*INT_TO_DINT(iEntrMilimetro18))/dMilimetro;
dSaidaPulso19:=(dPulso*INT_TO_DINT(iEntrMilimetro19))/dMilimetro;
dSaidaPulso20:=(dPulso*INT_TO_DINT(iEntrMilimetro20))/dMilimetro;

(* ---- MonitoraEncoder.fb.st ---- *)
FUNCTION_BLOCK MonitoraEncoder
VAR_INPUT
	xEncoHabilitado: BOOL;
	bResetAlmGeral: BOOL;
	dValorEncoder: DINT;
	tTempoCheck: TIME;
END_VAR
VAR_OUTPUT
	xAlarmeEncoder: BOOL;
	xAlarmeSonoro: BOOL;
	xEncoderOk: BOOL;
END_VAR
VAR
	TonCheck: TON;
	PassoEncoder: INT;
	dEncoder: DINT;
	dEncoderMenos: DINT;
	dEncoderMais: DINT;
	xCheckEnco: BOOL;
	xEncoderParado: BOOL;
	TonAlarme: TON;
	xTonAlarmeIn: BOOL;
	xTonAlarmeQ: BOOL;
	TonSinAlarme: TON;
	TonSinAlarmeIn: BOOL;
	TonSinAlarmePt: TIME;
	TonSinAlarmeQ: BOOL;
	TpSireneAlarme: TP;
	TpSireneAlarmeIn: BOOL;
	TpSireneAlarmePt: TIME;
	TpSireneAlarmeQ: BOOL;
END_VAR

TonCheck(IN:= NOT xCheckEnco , PT:=tTempoCheck , Q=>xCheckEnco , ET=> );

CASE PassoEncoder OF

	0: 	IF xCheckEnco AND xEncoHabilitado THEN
			PassoEncoder:=5;
		END_IF

	5:	//xTonAlarmeIn:=TRUE;
		//IF xTonAlarmeQ THEN
			PassoEncoder:=6;
		//END_IF

	6:	//xTonAlarmeIn:=FALSE;
		dEncoderMenos:=dEncoder-10;
		dEncoderMais:=dEncoder+10;
		PassoEncoder:=7;

	7:	IF dValorEncoder>=dEncoderMenos AND dValorEncoder<=dEncoderMais THEN
			xEncoderParado:=TRUE;
			xTonAlarmeIn:=TRUE;
			IF xTonAlarmeQ THEN
				xAlarmeEncoder:=TRUE;
				xEncoderOk:=FALSE;
				PassoEncoder:=20;
			END_IF
		ELSE
			xEncoderParado:=FALSE;
			xTonAlarmeIn:=FALSE;
			xEncoderOk:=true;
			PassoEncoder:=15;
		END_IF

	8: xEncoderParado:=TRUE;

	15:	dEncoder:=dValorEncoder;
		PassoEncoder:=0;

	20: IF bResetAlmGeral THEN
			xAlarmeEncoder:=FALSE;
			xAlarmeSonoro:=FALSE;
			PassoEncoder:=0;
		END_IF

END_CASE

TonAlarme (IN := xTonAlarmeIn,
           PT := T#500MS,
           Q => xTonAlarmeQ);

(*--- Alarme Sonoro ---*)
TpSireneAlarmeIn:=xAlarmeEncoder;

TpSireneAlarme (IN := TpSireneAlarmeIn,
                PT := T#500ms,
                Q => TpSireneAlarmeQ);

if TpSireneAlarmeQ then
	xAlarmeSonoro:=true;
end_if;

IF bResetAlmGeral THEN
	xAlarmeSonoro:=FALSE;
END_IF

(* ---- Patamar.fb.st ---- *)
FUNCTION_BLOCK Patamar
VAR_IN_OUT
	xIniciaPatamar: BOOL;
	xFimPatamar: BOOL;
	xResetBloco: BOOL;
END_VAR
VAR_INPUT
	rTemopar: REAL;
	rPatamar: REAL;
	rHisterese: REAL;
	rTempoPatamar: REAL;
	xDesabilitaZn: BOOL;
END_VAR
VAR_OUTPUT
	xSaida: BOOL;
	wStatusPatamar: WORD;
	rTempoPatamarDecorrido: REAL;
	rTempoPatamarRestante: REAL;
	rTempoFinal: REAL;
END_VAR
VAR
	PassoPatamar: INT;
	ControleTemperatura: FB_2points;
	stParametros: stPtPara;
	TempoPatamar: TON;
	TempoPatamarIn: BOOL;
	TempoPatamarQ: BOOL;
	TempoPatamarPt: TIME;
	TempoPatamarEt: TIME;
	tTempoCiclo: TIME;
	rTempoPatamarDecor: REAL;
END_VAR

CASE PassoPatamar OF

	0:	IF xIniciaPatamar THEN
			PassoPatamar:=5;
		END_IF

	5:	xIniciaPatamar:=FALSE;
		IF (rTempoPatamar=0) (*OR (rTemopar > (rPatamar+5))*) OR xDesabilitaZn THEN
			PassoPatamar:=10;
		ELSE
			ControleTemperatura.i_xEn:=TRUE;
			wStatusPatamar:=1;
			TempoPatamarIn:=TRUE;
			TempoPatamarPt:=REAL_TO_TIME (rTempoPatamar*1000);
			IF TempoPatamarQ THEN
				PassoPatamar:=10;
			END_IF
		END_IF

	10:	rTempoFinal:=rTempoPatamarDecor;
		PassoPatamar:=15;

	15:	xFimPatamar:=TRUE;
		wStatusPatamar:=2;
		TempoPatamarIn:=FALSE;
		ControleTemperatura.i_xEn:=FALSE;
		//PassoPatamar:=0;

END_CASE
TempoPatamar(IN:=TempoPatamarIn , PT:=TempoPatamarPt , Q=>TempoPatamarQ , ET=>TempoPatamarEt );
rTempoPatamarDecor:=(TIME_TO_REAL(TempoPatamarEt))/1000;
rTempoPatamarDecorrido:=rTempoPatamarDecor+(rTempoFinal);
rTempoPatamarRestante:=rTempoPatamar-rTempoPatamarDecorrido;

stParametros.rHyst:=	rHisterese;
stParametros.tCyclTime:=tTempoCiclo:=T#100MS;

ControleTemperatura(
	i_xEn:= ,
	i_rSp:= 		rPatamar,
	i_rActVal:= 	rTemopar,
	i_xManVal:= ,
	i_xManMode:= ,
	i_stPara:= 		stParametros,
	i_xErrRst:= ,
	q_xEn=> ,
	q_xBusy=> ,
	q_xOput=> 		xSaida,
	q_xErr=> ,
	q_uiErrId=> );

IF xResetBloco THEN
	xIniciaPatamar	:=FALSE;
	xFimPatamar		:=FALSE;
	//xResetBloco		:=FALSE;
	wStatusPatamar	:=0;
	TempoPatamarIn	:=FALSE;
	ControleTemperatura.i_xEn:=FALSE;
	PassoPatamar	:=0;
	rTempoFinal		:=0;
END_IF

(* ---- PidPwm.fb.st ---- *)
FUNCTION_BLOCK PidPwm
VAR_INPUT
	xLigaDesliga: BOOL;
	xHabilitaControle: BOOL;
	xForceResistencia: BOOL;
	xHabilitaResistencia: BOOL;
	AlarmeResistencia: BOOL;
	xRstTemperaturaOk: BOOL;
	xFornoComCarga: BOOL;
	rTermoparLeitura: REAL;
	rTermoparControle: REAL;
	rSetTemperatura: REAL;
	rProcentagem: REAL;
	rGanhoPorporcionaKp: REAL;
	rGanhoIntegralKi: REAL;
	rGanhoDerivativoKd: REAL;
	rTempoCiclo: REAL;
	xresetPidBlk:BOOL;
END_VAR
VAR_OUTPUT
	SaidaPwm: BOOL;
	xTemperaturaOk: BOOL;
	rTemperatura: REAL;
END_VAR
VAR
	PID: FB_PID;
	PWM: FB_PWM;
	rPidSaida: REAL;
	rPwmEntrada: REAL;
	xPwmSaida: BOOL;
	xTemperaturaExcesso: BOOL;
	tTempoCiclo: TIME;
END_VAR

PID.i_stPid.rLowLim:=0;
PID.i_stPid.rHighLim:=100;
PID.i_stPid.rTargCyclTime:=rTempoCiclo;
PID(
	i_xEn:= 		xHabilitaControle,
	i_rSp:= 		rSetTemperatura,
	i_rPv1:= 		rTermoparControle,
	i_iPv2:= 		,
	i_xHold:= 		,
	i_rKp:= 		rGanhoPorporcionaKp,
	i_rTn:= 		rGanhoIntegralKi,
	i_rTv:= 		rGanhoDerivativoKd,
	i_rTd:= 		210,
	i_xManMode:= 	,
	i_rManVal:= 	,
	i_stPid:= 		,
	i_xErrRst:= 	xresetPidBlk,
	q_xEn=> 		,
	q_xBusy=> 		,
	q_rPidOput=> 	rPidSaida,
	q_xMinLimActv=> ,
	q_xMaxLimActv=> ,
	q_xARWActv=> 	,
	q_xErr=> 		,
	q_uiErrId=> 	,
	q_sErrMsge=> 	,
	q_sFBstat=> 	);

rPwmEntrada:= rPidSaida*(rProcentagem/100);

tTempoCiclo:= REAL_TO_TIME (rTempoCiclo);
PWM.i_stPara.tCyclTime:=tTempoCiclo;
PWM.i_stPara.tPwmPeriod:=T#1000MS;
PWM(
	i_xEn:= 	xHabilitaControle,
	i_rIput:= 	rPwmEntrada,
	i_stPara:= 	,
	i_xErrRst:= xresetPidBlk,
	q_xEn=> 	,
	q_xBusy=> 	,
	q_xPstv=> 	xPwmSaida,
	q_xNgtv=> 	,
	q_xErr=> 	,
	q_uiErrId=> );

// Temperatura Atingiu Limite de 750 graus

IF (rTemperatura>=rSetTemperatura+50) AND xFornoComCarga THEN
	xTemperaturaExcesso:=TRUE;
ELSE
	xTemperaturaExcesso:=FALSE;
END_IF

SaidaPwm:= (xLigaDesliga AND xHabilitaResistencia AND NOT AlarmeResistencia  AND NOT xTemperaturaExcesso AND xPwmSaida) OR xForceResistencia;
rTemperatura:=rTermoparLeitura;

// Temeratura atingiu Set Point
IF (rTemperatura>=rSetTemperatura) AND xFornoComCarga THEN
	xTemperaturaOk:=TRUE;
END_IF
IF xRstTemperaturaOk OR NOT xFornoComCarga THEN
	xTemperaturaOk:=FALSE;
END_IF

(* ---- PidPwm_ONOFF.fb.st ---- *)
FUNCTION_BLOCK PidPwm_ONOFF
VAR_INPUT
	xLigaDesliga: BOOL;
	xHabilitaControle: BOOL;
	xForceResistencia: BOOL;
	xHabilitaResistencia: BOOL;
	AlarmeResistencia: BOOL;
	xRstTemperaturaOk: BOOL;
	xFornoComCarga: BOOL;
	rTermoparLeitura: REAL;
	rTermoparControle: REAL;
	rSetTemperatura: REAL;
	rProcentagem: REAL;
	rGanhoPorporcionaKp: REAL;
	rGanhoIntegralKi: REAL;
	rGanhoDerivativoKd: REAL;
	rTempoCiclo: REAL;
	xresetPidBlk:BOOL;
END_VAR
VAR_OUTPUT
	SaidaPwm: BOOL;
	xTemperaturaOk: BOOL;
	rTemperatura: REAL;
END_VAR
VAR
	///PID: FB_PID;
	///PWM: FB_PWM;
	rPidSaida: REAL;
	rPwmEntrada: REAL;
	xPwmSaida: BOOL;
	xTemperaturaExcesso: BOOL;
	TgPorcent: TimerGenerationPorc;
	rPorcentagemOn: REAL;
	rPorcentagemOff: REAL;
	tTimeOn: TIME;
	tTimeOff: TIME;
	TgPorcentOut: BOOL;
	xPwmSaidaOnOff: BOOL;
END_VAR

IF rSetTemperatura>=rTermoparControle AND xHabilitaControle THEN
	xPwmSaidaOnOff:=TRUE;
ELSE
	xPwmSaidaOnOff:=FALSE;
END_IF

rPorcentagemOn:=rProcentagem;
rPorcentagemOff:=100-rProcentagem;

tTimeOn:=REAL_TO_TIME (rPorcentagemOn)*10;
tTimeOff:=REAL_TO_TIME (rPorcentagemOff)*10;

TgPorcent(ENABLE:=xPwmSaidaOnOff , TIMELOW:= tTimeOn, TIMEHIGH:= tTimeOff, rPorceta:= rProcentagem, OUT=>TgPorcentOut );

xPwmSaida:=(TgPorcentOut);

SaidaPwm:= (xLigaDesliga AND xHabilitaResistencia AND NOT AlarmeResistencia  AND NOT xTemperaturaExcesso AND xPwmSaida) OR xForceResistencia;
rTemperatura:=rTermoparLeitura;

// Temperatura Atingiu Limite de 750 graus

IF (rTemperatura>=rSetTemperatura+50) AND xFornoComCarga THEN
	xTemperaturaExcesso:=TRUE;
ELSE
	xTemperaturaExcesso:=FALSE;
END_IF

// Temeratura atingiu Set Point
IF (rTemperatura>=rSetTemperatura) AND xFornoComCarga THEN
	xTemperaturaOk:=TRUE;
END_IF
IF xRstTemperaturaOk OR NOT xFornoComCarga THEN
	xTemperaturaOk:=FALSE;
END_IF

(* ---- PulsoConversorMm.fb.st ---- *)
FUNCTION_BLOCK PulsoConversorMm
VAR_INPUT
	dPulso: DINT;
	dMilimetro: DINT;
	dEntradaPulso01: DINT;
	dEntradaPulso02: DINT;
	dEntradaPulso03: DINT;
	dEntradaPulso04: DINT;
	dEntradaPulso05: DINT;
	dEntradaPulso06: DINT;
	dEntradaPulso07: DINT;
	dEntradaPulso08: DINT;
	dEntradaPulso09: DINT;
	dEntradaPulso10: DINT;
	dEntradaPulso11: DINT;
	dEntradaPulso12: DINT;
	dEntradaPulso13: DINT;
	dEntradaPulso14: DINT;
	dEntradaPulso15: DINT;
	dEntradaPulso16: DINT;
	dEntradaPulso17: DINT;
	dEntradaPulso18: DINT;
	dEntradaPulso19: DINT;
	dEntradaPulso20: DINT;
END_VAR
VAR_OUTPUT
	iSaidaMilimetro01: INT;
	iSaidaMilimetro02: INT;
	iSaidaMilimetro03: INT;
	iSaidaMilimetro04: INT;
	iSaidaMilimetro05: INT;
	iSaidaMilimetro06: INT;
	iSaidaMilimetro07: INT;
	iSaidaMilimetro08: INT;
	iSaidaMilimetro09: INT;
	iSaidaMilimetro10: INT;
	iSaidaMilimetro11: INT;
	iSaidaMilimetro12: INT;
	iSaidaMilimetro13: INT;
	iSaidaMilimetro14: INT;
	iSaidaMilimetro15: INT;
	iSaidaMilimetro16: INT;
	iSaidaMilimetro17: INT;
	iSaidaMilimetro18: INT;
	iSaidaMilimetro19: INT;
	iSaidaMilimetro20: INT;
END_VAR

iSaidaMilimetro01:=DINT_TO_INT((dEntradaPulso01*dMilimetro)/dPulso);
iSaidaMilimetro02:=DINT_TO_INT((dEntradaPulso02*dMilimetro)/dPulso);
iSaidaMilimetro03:=DINT_TO_INT((dEntradaPulso03*dMilimetro)/dPulso);
iSaidaMilimetro04:=DINT_TO_INT((dEntradaPulso04*dMilimetro)/dPulso);
iSaidaMilimetro05:=DINT_TO_INT((dEntradaPulso05*dMilimetro)/dPulso);
iSaidaMilimetro06:=DINT_TO_INT((dEntradaPulso06*dMilimetro)/dPulso);
iSaidaMilimetro07:=DINT_TO_INT((dEntradaPulso07*dMilimetro)/dPulso);
iSaidaMilimetro08:=DINT_TO_INT((dEntradaPulso08*dMilimetro)/dPulso);
iSaidaMilimetro09:=DINT_TO_INT((dEntradaPulso09*dMilimetro)/dPulso);
iSaidaMilimetro10:=DINT_TO_INT((dEntradaPulso10*dMilimetro)/dPulso);
iSaidaMilimetro11:=DINT_TO_INT((dEntradaPulso11*dMilimetro)/dPulso);
iSaidaMilimetro12:=DINT_TO_INT((dEntradaPulso12*dMilimetro)/dPulso);
iSaidaMilimetro13:=DINT_TO_INT((dEntradaPulso13*dMilimetro)/dPulso);
iSaidaMilimetro14:=DINT_TO_INT((dEntradaPulso14*dMilimetro)/dPulso);
iSaidaMilimetro15:=DINT_TO_INT((dEntradaPulso15*dMilimetro)/dPulso);
iSaidaMilimetro16:=DINT_TO_INT((dEntradaPulso16*dMilimetro)/dPulso);
iSaidaMilimetro17:=DINT_TO_INT((dEntradaPulso17*dMilimetro)/dPulso);
iSaidaMilimetro18:=DINT_TO_INT((dEntradaPulso18*dMilimetro)/dPulso);
iSaidaMilimetro19:=DINT_TO_INT((dEntradaPulso19*dMilimetro)/dPulso);
iSaidaMilimetro20:=DINT_TO_INT((dEntradaPulso20*dMilimetro)/dPulso);

(* ---- PulsoNegativo.fb.st ---- *)
FUNCTION_BLOCK PulsoNegativo
VAR_INPUT
	Entrada: BOOL;
END_VAR
VAR_OUTPUT
	SaidaPulsoNe: BOOL;
END_VAR
VAR
	Auxiliar: BOOL;
END_VAR

SaidaPulsoNe:= NOT Entrada AND NOT Auxiliar ;
Auxiliar:= NOT Entrada ;

(* ---- PulsoPositivo.fb.st ---- *)
FUNCTION_BLOCK PulsoPositivo
VAR_INPUT
	Entrada: BOOL;
END_VAR
VAR_OUTPUT
	SaidaPulsoPo: BOOL;
END_VAR
VAR
	Auxiliar: BOOL;
END_VAR

SaidaPulsoPo:= Entrada AND NOT Auxiliar ;
Auxiliar:= Entrada ;

(* ---- Rampa.fb.st ---- *)
FUNCTION_BLOCK Rampa
VAR_IN_OUT
	xIniciaRampa: BOOL;
	xFimRampa: BOOL;
	xResetBloco: BOOL;
END_VAR
VAR_INPUT
	rTemopar: REAL;
	rTempMedia: REAL;
	rPatamar: REAL;
	rTempoRampa: REAL;
	xDesabilitaZn: BOOL;
	xFimTotRampa: BOOL;
END_VAR
VAR_OUTPUT
	xSaida: BOOL;
	wStatusRampa: WORD;
	rTempoRampaDecorrido: REAL;
	rTempoRampaRestante: REAL;
	rTempoFinal: REAL;
	rSpTemperaturaUp: REAL;
END_VAR
VAR
	rSomaDegrau: REAL;
	PassoRampa: INT;
	PassoRampaInto: INT;
	TempoRealRampa: TON;
	TempoRealRampaIn: BOOL;
	TempoRealRampaPt: TIME;
	TempoRealRampaQ: BOOL;
	TempoRealRampaEt: TIME;
	TempoIntegracao: TON;
	TempoIntegracaoIn: BOOL;
	TempoIntegracaoPt: TIME;
	TempoIntegracaoQ: BOOL;
	TempoIntegracaoEt: TIME;
	TempoCiclo: TON;
	TempoCicloIn: BOOL;
	TempoCicloPt: TIME;
	TempoCicloQ: BOOL;
	TempoCicloEt: TIME;
	rDegrau: REAL;
	rDxTemperatura: REAL;
	rTempoIntegracao: REAL;
	tTempoCiclo: TIME := TIME#100ms;
	xIniciaTempoCiclo: BOOL;
	rTempoRampaDecor: REAL;
	tTempoIntegracao: TIME;
	rDxTempoIntegracao: REAL;
	rDxTempoRampa: REAL;
	rTempoSubCiclo: REAL;
END_VAR

TempoRealRampaPt:=REAL_TO_TIME((rTempoRampa+((rTempoRampa*20)/100))*1000);

CASE PassoRampa OF

	0: IF xIniciaRampa THEN
			PassoRampa:=1;
	   END_IF

	1: 	xIniciaRampa:=FALSE;
		IF (rTemopar < rPatamar) OR xDesabilitaZn THEN
			wStatusRampa:=1;
			TempoRealRampaIn:=TRUE;
			rDegrau:=0.1;
			rDxTemperatura:= rPatamar-rTemopar;
			PassoRampa:=2;
		ELSE
		PassoRampa:=10;
		END_IF

	2:	rDxTempoRampa:=((rTempoRampa)*0.1);
		rTempoIntegracao:=rDxTempoRampa/rDxTemperatura;
	   	PassoRampa:=3;

	3:rSpTemperaturaUp:=rTemopar;
	   PassoRampa:=4;

	4: xSaida:=TRUE;
		PassoRampa:=5;

	5:	IF rSpTemperaturaUp <= rPatamar AND NOT xDesabilitaZn THEN
			rSpTemperaturaUp:=rSpTemperaturaUp+rDegrau;
			PassoRampa:=6;
		ELSE
			PassoRampa:=10;
		END_IF;

	6: TempoIntegracaoIn:=TRUE;
		rDxTempoIntegracao:=(rTempoIntegracao*1000);
		rTempoSubCiclo:=rDxTempoIntegracao-50;
		tTempoIntegracao:=REAL_TO_TIME (rTempoSubCiclo);
	 	TempoIntegracaoPt:=tTempoIntegracao;
		IF NOT TempoIntegracaoQ THEN
				CASE PassoRampaInto OF

					0:	xIniciaTempoCiclo:=TRUE;
						PassoRampaInto:=2;

					2:	xIniciaTempoCiclo:=FALSE;
						TempoCicloIn:=TRUE;
						TempoCicloPt:=tTempoCiclo;
						IF TempoIntegracaoQ THEN
		   					PassoRampaInto:=3;
	   					END_IF

					3:	TempoCicloIn:=FALSE;
						IF rTemopar< rSpTemperaturaUp THEN
							PassoRampaInto:=4;
						END_IF
						IF rTemopar >= rSpTemperaturaUp THEN
							PassoRampaInto:=5;
						END_IF
						//IF rTemopar >= rPatamar THEN
						//	PassoRampa:=10;
						//END_IF

					4:	xSaida:=TRUE;
						IF rTempoRampaRestante <=10 THEN
							PassoRampa:=12;
						ELSE
							PassoRampaInto:=0;
						END_IF
						//PassoRampaInto:=0;

					5:	xSaida:=FALSE;
						PassoRampaInto:=0;

				END_CASE
		END_IF

	   	IF TempoIntegracaoQ THEN
		   	PassoRampa:=7;
			rSomaDegrau:=rSomaDegrau+rDegrau;
			//PassoRampa:=5;
	   	END_IF

	7: TempoIntegracaoIn:=FALSE;
		IF rTempoRampaRestante <=10 THEN
			PassoRampa:=12;
		ELSE
			IF rTemopar< rSpTemperaturaUp THEN
				PassoRampa:=8;
			END_IF
			IF rTemopar >= rSpTemperaturaUp THEN
				PassoRampa:=9;
			END_IF
			IF (*rTempMedia*)rTemopar  >= rPatamar THEN
				PassoRampa:=10;
			END_IF
		END_IF

	12:	IF ((*rTempMedia*)rTemopar < rPatamar) AND NOT xDesabilitaZn THEN
			xSaida:=TRUE;
		END_IF
		IF	((*rTempMedia*)rTemopar >= rPatamar) AND NOT xDesabilitaZn THEN
			PassoRampa:=10;
		END_IF
		IF xDesabilitaZn THEN
			PassoRampa:=10;
		END_IF

	8:	xSaida:=TRUE;
		PassoRampa:=5;

	9:	xSaida:=FALSE;
		PassoRampa:=5;

	10:	xSaida:=FALSE;
		rTempoFinal:=rTempoRampaDecor;
		PassoRampa:=11;

	11:	xFimRampa:=TRUE;
		wStatusRampa:=2;
		TempoRealRampaIn:=FALSE;
		IF (rTemopar < rPatamar) AND NOT xDesabilitaZn THEN
			xSaida:=TRUE;
		ELSE
			xSaida:=FALSE;
		END_IF
		IF xFimTotRampa THEN
			PassoRampa:=20;
		END_IF

	20: xSaida:=FALSE;

		//PassoRampaInto:=0;

END_CASE
TempoIntegracao(IN:=TempoIntegracaoIn , PT:=TempoIntegracaoPt , Q=>TempoIntegracaoQ , ET=> );
TempoRealRampa(IN:=TempoRealRampaIn , PT:=TempoRealRampaPt , Q=> , ET=>TempoRealRampaEt );
rTempoRampaDecor:=(TIME_TO_REAL(TempoRealRampaEt))/1000;
rTempoRampaRestante:=rTempoRampa-rTempoRampaDecorrido;

rTempoRampaDecorrido:=rTempoRampaDecor+(rTempoFinal);

IF xResetBloco THEN
	xIniciaRampa	:=FALSE;
	xFimRampa		:=FALSE;
	//xResetBloco		:=FALSE;
	wStatusRampa	:=0;
	xSaida			:=FALSE;
	TempoRealRampaIn:=FALSE;
	TempoIntegracaoIn:=FALSE;
	TempoCicloIn	:=FALSE;
	PassoRampa		:=0;
	PassoRampaInto	:=0;
	rTempoFinal		:=0;
END_IF

(* ---- RampaCiclo.fb.st ---- *)
FUNCTION_BLOCK RampaCiclo
VAR_INPUT
	iTermopar	: INT ;
	rSpTemperatura	: REAL ;
	iTempoEstab	: INT ;
	xReset		: BOOL ;
END_VAR
VAR_OUTPUT
	xStartRampaCiclo	: BOOL ;
	xRampaAtiva	: BOOL ;
	TemperUp	: BOOL ;
	TemperDown	: BOOL ;
	rSpTemperaturaUp	: REAL ;
	rSetTemperaturaRampa: REAL ;
END_VAR
VAR
	iDadoEntrada: INT ;
	iDadoSaida	: INT ;

	rTermopar	: REAL ;

	rTempoInicialRamp : REAL ;
	rTempoFinalRamp: REAL ;
	rTempoRamp	: REAL ;

	rTemperaturaRampIni: REAL ;
	rTemperaturaRampFim: REAL ;

	rTamperaturaRamp	: REAL ;
	rGradienteRamp		:REAL ;

	rTempoTemperatura: REAL ;
	rTempoTemperaturaSp: REAL ;

	TgTemper : TimerGeneration;

	PulsoEntrada: PulsoPositivo;
	xPulsoEntrada: BOOL ;
	xPulsoSaida	: BOOL;

	TonDlyCarga	: TON ;
	xTonDlyCargaIn	: BOOL ;
	xTonDlyCargaQ	: BOOL ;
	tTonDlyCargaPt	: BOOL ;

	PulsoStartRampa : PulsoPositivo ;
	xPulsoStartRampa: BOOL ;

	TonCicloRamp	: TON ;
	xTonCicloRampIn	: BOOL ;
	xTonCicloRampQ	: BOOL ;

	rTemperaturaSpRampOk	: BOOL;
	rTemperaturaRampOk	: BOOL;
	rTempoRampOk 	: BOOL;

	bloqSpR: BOOL;
	bloqR: BOOL;
END_VAR

// Teste Aquecimento Rampa

rTermopar:=INT_TO_REAL(iTermopar/10);

iDadoEntrada:=	iTermopar;

TgTemper(ENABLE:= TRUE, TIMELOW:= T#500MS, TIMEHIGH:=T#500MS , OUT=> xPulsoEntrada);

PulsoEntrada(Entrada:=xPulsoEntrada , SaidaPulsoPo=> xPulsoSaida);

	IF xPulsoSaida THEN
		iDadoSaida:=iDadoEntrada;
		iDadoEntrada:=iTermopar;
	END_IF

	IF 	iDadoSaida<iTermopar THEN
		TemperUp:=TRUE;
		TemperDown:=FALSE;
	END_IF

	IF 	iDadoSaida>iTermopar THEN
		TemperUp:=FALSE;
		TemperDown:=TRUE;
	END_IF

(*IF xReset THEN
	iDadoSaida:=0;
END_IF*)

xTonDlyCargaIn:=xFornoCheio;
TonDlyCarga(IN:= xTonDlyCargaIn, PT:=T#15S , Q=> xTonDlyCargaQ, ET=> );

IF xTonDlyCargaQ AND TemperUp THEN
	xStartRampaCiclo:=TRUE;
END_IF

IF NOT xFornoCheio THEN
	xStartRampaCiclo:=FALSE;
	xRampaAtiva	:= FALSE ;
END_IF

PulsoStartRampa(Entrada:= xStartRampaCiclo, SaidaPulsoPo=> xPulsoStartRampa);

IF xPulsoStartRampa THEN
	rTempoInicialRamp:=INT_TO_REAL(iTempoAquecFornoDecorrido);
	rTempoFinalRamp:=INT_TO_REAL(iTempoAquecimForno-iTempoEstab);
	rTemperaturaRampIni:=rTermopar;
	rTemperaturaRampFim:=rSpTemperatura;
	rSpTemperaturaUp:=rTemperaturaRampIni;
	xRampaAtiva	:= TRUE ;
	bloqSpR:=FALSE;
	bloqR:=FALSE;
END_IF

rTempoRamp:=rTempoFinalRamp-rTempoInicialRamp;
rTamperaturaRamp:=rTemperaturaRampFim-rTemperaturaRampIni;

rGradienteRamp:=rTamperaturaRamp/rTempoRamp;

xTonCicloRampIn := NOT xTonCicloRampQ AND xStartRampaCiclo ;
TonCicloRamp(IN:= xTonCicloRampIn, PT:=T#940MS , Q=> xTonCicloRampQ, ET=> );
IF xTonCicloRampQ AND rSpTemperaturaUp<=rSpTemperatura THEN
	rSpTemperaturaUp:=rSpTemperaturaUp+rGradienteRamp;
END_IF

IF rSpTemperaturaUp >= rSpTemperatura THEN rTemperaturaSpRampOk :=TRUE; ELSE rTemperaturaSpRampOk :=FALSE; END_IF
IF 	rTempoFinalRamp <= iTempoAquecFornoDecorrido THEN rTempoRampOk:=TRUE ; ELSE rTempoRampOk:=FALSE; END_IF
IF  rTermopar >= rSpTemperatura THEN rTemperaturaRampOk :=TRUE; ELSE rTemperaturaRampOk :=FALSE; END_IF

IF rTemperaturaSpRampOk AND NOT bloqSpR THEN
rTempoTemperaturaSp:=iTempoAquecFornoDecorrido;
bloqSpR:=TRUE;
END_IF
IF rTemperaturaRampOk AND NOT bloqR THEN
rTempoTemperatura:=iTempoAquecFornoDecorrido;
xRampaAtiva	:= FALSE ;
bloqR:=TRUE;
END_IF

IF xStartRampaCiclo THEN
	rSetTemperaturaRampa:=rSpTemperaturaUp;
//	xReleSsrSuperior[24]:=xReleSsrSuperiorRampa;
ELSE
	rSetTemperaturaRampa:=rSpTemperatura;
//	xReleSsrSuperior[24]:=Q_xAquecimentoPwm;
END_IF

// Liga/Desliga Resistência
(*IF rSetTemperaturaRampa>=rTermopar THEN
		xReleSsrSuperiorRampa:=TRUE;
ELSE
		xReleSsrSuperiorRampa:=FALSE;
END_IF*)

(* ---- Registrador.fb.st ---- *)
FUNCTION_BLOCK Registrador
VAR_INPUT
	xPulsoEntrada: BOOL;
	xReset: BOOL;
	iDadoEntrada: INT;
END_VAR
VAR_OUTPUT
	iDadoSaida: INT;
END_VAR
VAR
	PulsoEntrada: PulsoPositivo;
	xPulsoSaida: BOOL;
END_VAR

PulsoEntrada(Entrada:=xPulsoEntrada , SaidaPulsoPo=> xPulsoSaida);

IF xPulsoSaida THEN
	iDadoSaida:=iDadoEntrada;
END_IF

IF xReset THEN
	iDadoSaida:=0;
END_IF

(* ---- RegistradorMedia.fb.st ---- *)
FUNCTION_BLOCK RegistradorMedia
VAR_INPUT
	rDadoEntrada: REAL;
END_VAR
VAR_OUTPUT
	rDadoSaida: REAL;
END_VAR
VAR
	Tg01: TimerGeneration;
	PulsoEntrada: PulsoPositivo;
	xPulsoEntrada: BOOL;
	xPulsoSaida: BOOL;
	rDadoAuxiliar01: REAL;
	rDadoAuxiliar02: REAL;
	rDadoAuxiliar03: REAL;
	rDadoAuxiliar04: REAL;
	rDadoAuxiliar05: REAL;
	rDadoAuxiliar06: REAL;
	rDadoAuxiliar07: REAL;
	rDadoAuxiliar08: REAL;
	rDadoAuxiliar09: REAL;
	rDadoAuxiliar10: REAL;
END_VAR

Tg01(ENABLE:= TRUE, TIMELOW:=T#1000MS , TIMEHIGH:=T#50MS , OUT=>xPulsoEntrada );
PulsoEntrada(Entrada:=xPulsoEntrada , SaidaPulsoPo=> xPulsoSaida);

IF xPulsoSaida THEN
	rDadoAuxiliar10:=rDadoAuxiliar09;
	rDadoAuxiliar09:=rDadoAuxiliar08;
	rDadoAuxiliar08:=rDadoAuxiliar07;
	rDadoAuxiliar07:=rDadoAuxiliar06;
	rDadoAuxiliar06:=rDadoAuxiliar05;
	rDadoAuxiliar05:=rDadoAuxiliar04;
	rDadoAuxiliar04:=rDadoAuxiliar03;
	rDadoAuxiliar03:=rDadoAuxiliar02;
	rDadoAuxiliar02:=rDadoAuxiliar01;
	rDadoAuxiliar01:=rDadoEntrada;
END_IF

rDadoSaida:=( rDadoAuxiliar10 + rDadoAuxiliar09 + rDadoAuxiliar08 + rDadoAuxiliar07 + rDadoAuxiliar06 + rDadoAuxiliar05 + rDadoAuxiliar04 + rDadoAuxiliar03 + rDadoAuxiliar02 + rDadoAuxiliar01)/10;

(* ---- SelecaoEspessura.fb.st ---- *)
FUNCTION_BLOCK SelecaoEspessura
VAR_INPUT
	Selecao: BOOL;
	Entrada01: INT;
	Entrada02: INT;
END_VAR
VAR_OUTPUT
	Saida: INT;
END_VAR

IF Selecao THEN
	Saida:=Entrada01;
ELSE
	Saida:=Entrada02;
END_IF

(* ---- Sr10.fb.st ---- *)
FUNCTION_BLOCK Sr10
VAR_INPUT
	xPulsoRegistro: BOOL;
	xPulsoReset: BOOL;
	iDadoEntrada01: INT;
	iDadoEntrada02: INT;
	iDadoEntrada03: INT;
	iDadoEntrada04: INT;
	iDadoEntrada05: INT;
	iDadoEntrada06: INT;
	iDadoEntrada07: INT;
	iDadoEntrada08: INT;
	iDadoEntrada09: INT;
	iDadoEntrada10: INT;
END_VAR
VAR_OUTPUT
	iDadoSaida01: INT;
	iDadoSaida02: INT;
	iDadoSaida03: INT;
	iDadoSaida04: INT;
	iDadoSaida05: INT;
	iDadoSaida06: INT;
	iDadoSaida07: INT;
	iDadoSaida08: INT;
	iDadoSaida09: INT;
	iDadoSaida10: INT;
END_VAR
VAR
	Registrador01: Registrador;
	Registrador02: Registrador;
	Registrador03: Registrador;
	Registrador04: Registrador;
	Registrador05: Registrador;
	Registrador06: Registrador;
	Registrador07: Registrador;
	Registrador08: Registrador;
	Registrador09: Registrador;
	Registrador10: Registrador;
END_VAR

Registrador01(xPulsoEntrada:=xPulsoRegistro , xReset:=xPulsoReset , iDadoEntrada:= iDadoEntrada01, iDadoSaida=> iDadoSaida01 );
Registrador02(xPulsoEntrada:=xPulsoRegistro , xReset:=xPulsoReset , iDadoEntrada:= iDadoEntrada02, iDadoSaida=> iDadoSaida02 );
Registrador03(xPulsoEntrada:=xPulsoRegistro , xReset:=xPulsoReset , iDadoEntrada:= iDadoEntrada03, iDadoSaida=> iDadoSaida03 );
Registrador04(xPulsoEntrada:=xPulsoRegistro , xReset:=xPulsoReset , iDadoEntrada:= iDadoEntrada04, iDadoSaida=> iDadoSaida04 );
Registrador05(xPulsoEntrada:=xPulsoRegistro , xReset:=xPulsoReset , iDadoEntrada:= iDadoEntrada05, iDadoSaida=> iDadoSaida05 );
Registrador06(xPulsoEntrada:=xPulsoRegistro , xReset:=xPulsoReset , iDadoEntrada:= iDadoEntrada06, iDadoSaida=> iDadoSaida06 );
Registrador07(xPulsoEntrada:=xPulsoRegistro , xReset:=xPulsoReset , iDadoEntrada:= iDadoEntrada07, iDadoSaida=> iDadoSaida07 );
Registrador08(xPulsoEntrada:=xPulsoRegistro , xReset:=xPulsoReset , iDadoEntrada:= iDadoEntrada08, iDadoSaida=> iDadoSaida08 );
Registrador09(xPulsoEntrada:=xPulsoRegistro , xReset:=xPulsoReset , iDadoEntrada:= iDadoEntrada09, iDadoSaida=> iDadoSaida09 );
Registrador10(xPulsoEntrada:=xPulsoRegistro , xReset:=xPulsoReset , iDadoEntrada:= iDadoEntrada10, iDadoSaida=> iDadoSaida10 );

(* ---- StatCircuitoResist.fb.st ---- *)
FUNCTION_BLOCK StatCircuitoResist
VAR_INPUT
	/// Valor acima do qual considera Resistência Ligada
	iAmpLigada: UINT;
	/// Valor da Leitura de Corrente Diretamente pelo Sensor
	iAmperagem: UINT;
	/// Acionamento do Rele de Estado Sólido
	xSaidaRele: BOOL;
	/// Retorno do Rele de Estado Sólido
	xRetorRele: BOOL;
END_VAR
VAR_OUTPUT
	/// Resistencia Ligada
	xLigada: BOOL;
	/// Resistência Desligada
	xDeslig: BOOL;
	/// Rele com Defeito Aberto ou Disjuntor Desligado
	xReleAb: BOOL;
	/// Rele com Defeito Fechado em Curto Circuito
	xReleCc: BOOL;
	/// Resistência Quebrada ou Fusível Aberto
	xResAbe: BOOL;
END_VAR

// Bloco de Identificação de Status dos Reles e Resistências

IF iAmperagem>=	iAmpLigada THEN
	xLigada:=TRUE;
	xDeslig:=FALSE;
ELSE
	xLigada:=FALSE;
	xDeslig:=TRUE;
END_IF

IF xDeslig AND xSaidaRele AND NOT xRetorRele THEN
	xReleAb:=TRUE;
ELSE
	xReleAb:=FALSE;
END_IF

IF xDeslig AND xSaidaRele AND xRetorRele THEN
	xResAbe:=TRUE;
ELSE
	xResAbe:=FALSE;
END_IF

IF xLigada AND NOT xSaidaRele THEN
	xReleCc:=TRUE;
ELSE
	xReleCc:=FALSE;
END_IF

(* ---- Temporizador.fb.st ---- *)
FUNCTION_BLOCK Temporizador
VAR_INPUT
	IniciaTempo: BOOL;
	AbortaTempo: BOOL;
	SetPointTempo: INT;
END_VAR
VAR_OUTPUT
	TempoDecorrido: INT;
	TempoRestante: INT;
END_VAR
VAR_IN_OUT
	FimTempo: BOOL;
END_VAR
VAR
	Ton01: TON;
	Ton01In: BOOL;
	Ton01Et: TIME;
	FimTempoAux: BOOL;
	TempoDecorridoAux: INT;
END_VAR

IF IniciaTempo AND NOT FimTempo THEN
	Ton01In:=TRUE;
END_IF

Ton01 (IN := Ton01In, PT := T#9999S, ET => Ton01Et);

IF  (DINT_TO_INT((TIME_TO_DINT(Ton01Et))/1000)>= SetPointTempo) AND Ton01In THEN
	FimTempoAux:=TRUE;
ELSE
	FimTempoAux:=FALSE;
END_IF

TempoDecorridoAux:= DINT_TO_INT((TIME_TO_DINT(Ton01Et))/1000);

IF NOT FimTempo THEN
	TempoDecorrido:=TempoDecorridoAux;
	TempoRestante:=SetPointTempo-TempoDecorrido;
END_IF

IF (FimTempoAux OR AbortaTempo) AND Ton01In THEN
	FimTempo:=TRUE;
	Ton01In:=FALSE;
END_IF

(* ---- TimerGeneration.fb.st ---- *)
FUNCTION_BLOCK TimerGeneration
VAR_INPUT
	ENABLE: BOOL;
	TIMELOW: TIME;
	TIMEHIGH: TIME;
END_VAR
VAR_OUTPUT
	OUT: BOOL;
END_VAR
VAR
	T1: TON;
	T1In: BOOL;
	T1Q: BOOL;
	T2: TON;
	T2In: BOOL;
	T2Q: BOOL;
END_VAR

T1In:= ENABLE AND NOT T2Q;
T1(IN:=T1In , PT:=TIMEHIGH , Q=>T1Q , ET=> );
T2In:=T1Q;
T2(IN:=T2In , PT:=TIMELOW , Q=>T2Q , ET=> );
OUT:=T1Q;

(* ---- TimerGenerationPorc.fb.st ---- *)
FUNCTION_BLOCK TimerGenerationPorc
VAR_INPUT
	ENABLE: BOOL;
	TIMELOW: TIME;
	TIMEHIGH: TIME;
	rPorceta: REAL;
END_VAR
VAR_OUTPUT
	OUT: BOOL;
END_VAR
VAR
	T1: TON;
	T1In: BOOL;
	T1Q: BOOL;
	T2: TON;
	T2In: BOOL;
	T2Q: BOOL;
END_VAR

T1In:= ENABLE AND NOT T2Q;

T1(IN:=T1In , PT:=TIMEHIGH , Q=>T1Q , ET=> );
T2In:=T1Q;

T2(IN:=T2In , PT:=TIMELOW , Q=>T2Q , ET=> );
OUT:=T1Q;

IF rPorceta = 0 THEN
	OUT:=0;
END_IF

IF (rPorceta >= 95) AND ENABLE THEN
	OUT:=1;
END_IF

(* ---- TrocaValor.fb.st ---- *)
FUNCTION_BLOCK TrocaValor
VAR_INPUT
	ValorNovo: REAL;
END_VAR
VAR_OUTPUT
	Saida: BOOL;
	ValorAtual: REAL;
END_VAR

IF ValorAtual<>ValorNovo THEN
	ValorAtual:=ValorNovo;
	Saida:=TRUE;
ELSE
	Saida:=FALSE;
END_IF

(* ---- WordBit.fb.st ---- *)
FUNCTION_BLOCK WordBit
VAR_INPUT
	uWord: UINT;
END_VAR
VAR_OUTPUT
	xbit0: BOOL;
	xbit1: BOOL;
	xbit2: BOOL;
	xbit3: BOOL;
	xbit4: BOOL;
	xbit5: BOOL;
	xbit6: BOOL;
	xbit7: BOOL;
	xbit8: BOOL;
	xbit9: BOOL;
	xbit10: BOOL;
	xbit11: BOOL;
	xbit12: BOOL;
	xbit13: BOOL;
	xbit14: BOOL;
	xbit15: BOOL;
END_VAR

xbit0:=uWord.0;
xbit1:=uWord.1;
xbit2:=uWord.2;
xbit3:=uWord.3;
xbit4:=uWord.4;
xbit5:=uWord.5;
xbit6:=uWord.6;
xbit7:=uWord.7;
xbit8:=uWord.8;
xbit9:=uWord.9;
xbit10:=uWord.10;
xbit11:=uWord.11;
xbit12:=uWord.12;
xbit13:=uWord.13;
xbit14:=uWord.14;
xbit15:=uWord.15;
